{attribute 'pack_mode' := '1'}
TYPE ST_Calibrate EXTENDS ST_MsgToPLC:
STRUCT
    (* TBD - calibration parameters. *)
END_STRUCT
END_TYPE

(* stored: Version 1.1.0.1, ProductVersion 3.1.4022.18
   DUT ST_Calibrate: Id {af3cc025-0115-4561-aba6-ee6446d98b19} *)
